PROGRAM Stationary_Load_State
VAR
END_VAR

IF Shuttle.LocationTrigger.Q THEN
	
	Stationary.LoadMismatchCheck	:= TRUE;
	
	IF Shuttle.Present THEN
		
		Stationary.IsLargeOrMedium	:= TRUE;
		Stationary.IsSmall			:= FALSE;
		
		IF Shuttle.LoadPresentCenter THEN
			
			Stationary.LoadPresent[1]	:= TRUE;
			Stationary.LoadPresent[2]	:= TRUE;
		
		ELSE
			
			Stationary.LoadPresent[1]	:= FALSE;
			Stationary.LoadPresent[2]	:= FALSE;
			
		END_IF
	
	ELSE
		
		Stationary.IsLargeOrMedium	:= FALSE;
		Stationary.IsSmall			:= TRUE;
	
		IF Shuttle.LoadPresent[1] THEN
			
			Stationary.LoadPresent[1]	:= TRUE;
			
		ELSE
			
			Stationary.LoadPresent[1]	:= FALSE;
		
		END_IF
		
		IF Shuttle.LoadPresent[2] THEN
			
			Stationary.LoadPresent[2]	:= TRUE;
			
		ELSE
			
			Stationary.LoadPresent[2]	:= FALSE;
		
		END_IF
		
	END_IF

END_IF

END_PROGRAM

(* stored: Version 1.1.0.1, ProductVersion 3.1.4024.9
   POU Stationary_Load_State: Id {a29863dd-b8a9-4ae7-8a05-c4d344874b05}, SpecialFunc None *)
